// TIA Portal V18 export
// export: Created 2025-12-01T17:51:29.9840395Z, ExportSetting None, DisplayName Totally Integrated Automation Portal, DisplayVersion V18 Update 5, DisplayName TIA Portal Openness, DisplayVersion V18 Update 5, DisplayName TIA Portal Teamcenter Gateway, DisplayVersion V18, DisplayName TIA Portal Version Control Interface, DisplayVersion V18, DisplayName STEP 7 Professional, DisplayVersion V18 Update 5, DisplayName STEP 7 Safety, DisplayVersion V18, DisplayName WinCC Professional, DisplayVersion V18 Update 5
DATA_BLOCK "PartData_Interface_DB"   // DB1500
{ S7_Optimized_Access := 'TRUE' }
// stored: MemoryReserve 100
   VAR
      PartDataID : Int := 1;   // 物料数据序号
      PartData { S7_SetPoint := 'True'} : Array[1..4] of "PartData_UDT";
      PartCMD : Array[1..4] of Struct
         Set : Bool;
         Use : Bool;
      END_STRUCT;
   END_VAR
BEGIN
   // PartData[1] : XXX物料
   // PartData[2] : XXX物料
   // PartData[3] : XXX物料
   // PartData[4] : XXX物料
END_DATA_BLOCK
